(* PLC project test_IXL.project, CODESYS CODESYS V3.5 SP20 *)
(* stored: creationDateTime 2024-11-21T22:24:16.9503373, modificationDateTime 2024-07-08T19:29:50.2349361 *)

PROGRAM PLC_PRG
  VAR
    TC_occupied_101 : BOOL;
    TC_occupied_103 : BOOL;
    TC_occupied_105 : BOOL;
    TC_occupied_107 : BOOL;
    TC_occupied_109 : BOOL;
    TC_occupied_111 : BOOL;
    TC_occupied_113 : BOOL;
    TC_occupied_115 : BOOL;
    TC_occupied_102 : BOOL;
    TC_occupied_104 : BOOL;
    TC_occupied_106 : BOOL;
    TC_occupied_108 : BOOL;
    TC_occupied_110 : BOOL;
    TC_occupied_112 : BOOL;
    TC_occupied_114 : BOOL;
    TC_occupied_116 : BOOL;
    switch_detected_left_01 : BOOL;
    switch_detected_right_01 : BOOL;
    switch_detected_left_02 : BOOL;
    switch_detected_right_02 : BOOL;
    route_destruction_demand_AB : BOOL;
    route_destruction_demand_BC : BOOL;
    route_destruction_demand_ED : BOOL;
    route_destruction_demand_CD : BOOL;
    route_destruction_demand_DC : BOOL;
    route_destruction_demand_CB : BOOL;
    route_formation_demand_AB : BOOL;
    route_formation_demand_BC : BOOL;
    route_formation_demand_ED : BOOL;
    route_formation_demand_CD : BOOL;
    route_formation_demand_DC : BOOL;
    route_formation_demand_CB : BOOL;
    switch_manual_override_01 : BOOL;
    switch_manual_override_02 : BOOL;
    signal_open_route_201 : BOOL;
    signal_open_route_203 : BOOL;
    signal_open_route_205 : BOOL;
    signal_open_route_206 : BOOL;
    signal_open_route_208 : BOOL;
    signal_open_block_201 : BOOL;
    signal_open_block_203 : BOOL;
    signal_open_block_205 : BOOL;
    signal_open_block_206 : BOOL;
    signal_open_block_208 : BOOL;
    signal_open_block_207 : BOOL;
    signal_open_block_204 : BOOL;
    signal_open_block_210 : BOOL;
    switch_command_left_01 : BOOL;
    switch_command_right_01 : BOOL;
    switch_command_left_02 : BOOL;
    switch_command_right_02 : BOOL;
    route_open_AB : BOOL;
    route_open_BC : BOOL;
    route_open_ED : BOOL;
    route_open_CD : BOOL;
    route_open_DC : BOOL;
    route_open_CB : BOOL;
    route_destruction_acq_AB : BOOL;
    route_destruction_acq_BC : BOOL;
    route_destruction_acq_ED : BOOL;
    route_destruction_acq_CD : BOOL;
    route_destruction_acq_DC : BOOL;
    route_destruction_acq_CB : BOOL;
    route_state_AB : route_state;
    route_state_BC : route_state;
    route_state_ED : route_state;
    route_state_CD : route_state;
    route_state_DC : route_state;
    route_state_CB : route_state;
  END_VAR
  VAR CONSTANT
    DELAY_DEST_DC : TIME := TIME#30s0ms;
    DELAY_DEST_CB : TIME := TIME#30s0ms;
    DELAY_DEST_ED : TIME := TIME#30s0ms;
    DELAY_DEST_CD : TIME := TIME#30s0ms;
    DELAY_DEST_BC : TIME := TIME#30s0ms;
    DELAY_DEST_AB : TIME := TIME#30s0ms;
  END_VAR
  VAR
    direction_lock_CB : BOOL;
    direction_lock_AB : BOOL;
  END_VAR
  VAR  (* added by the conversion: wires and edge detectors of the diagram *)
    _AND70000000008_OUT : BOOL;
    _AND80000000007_OUT : BOOL;
  END_VAR

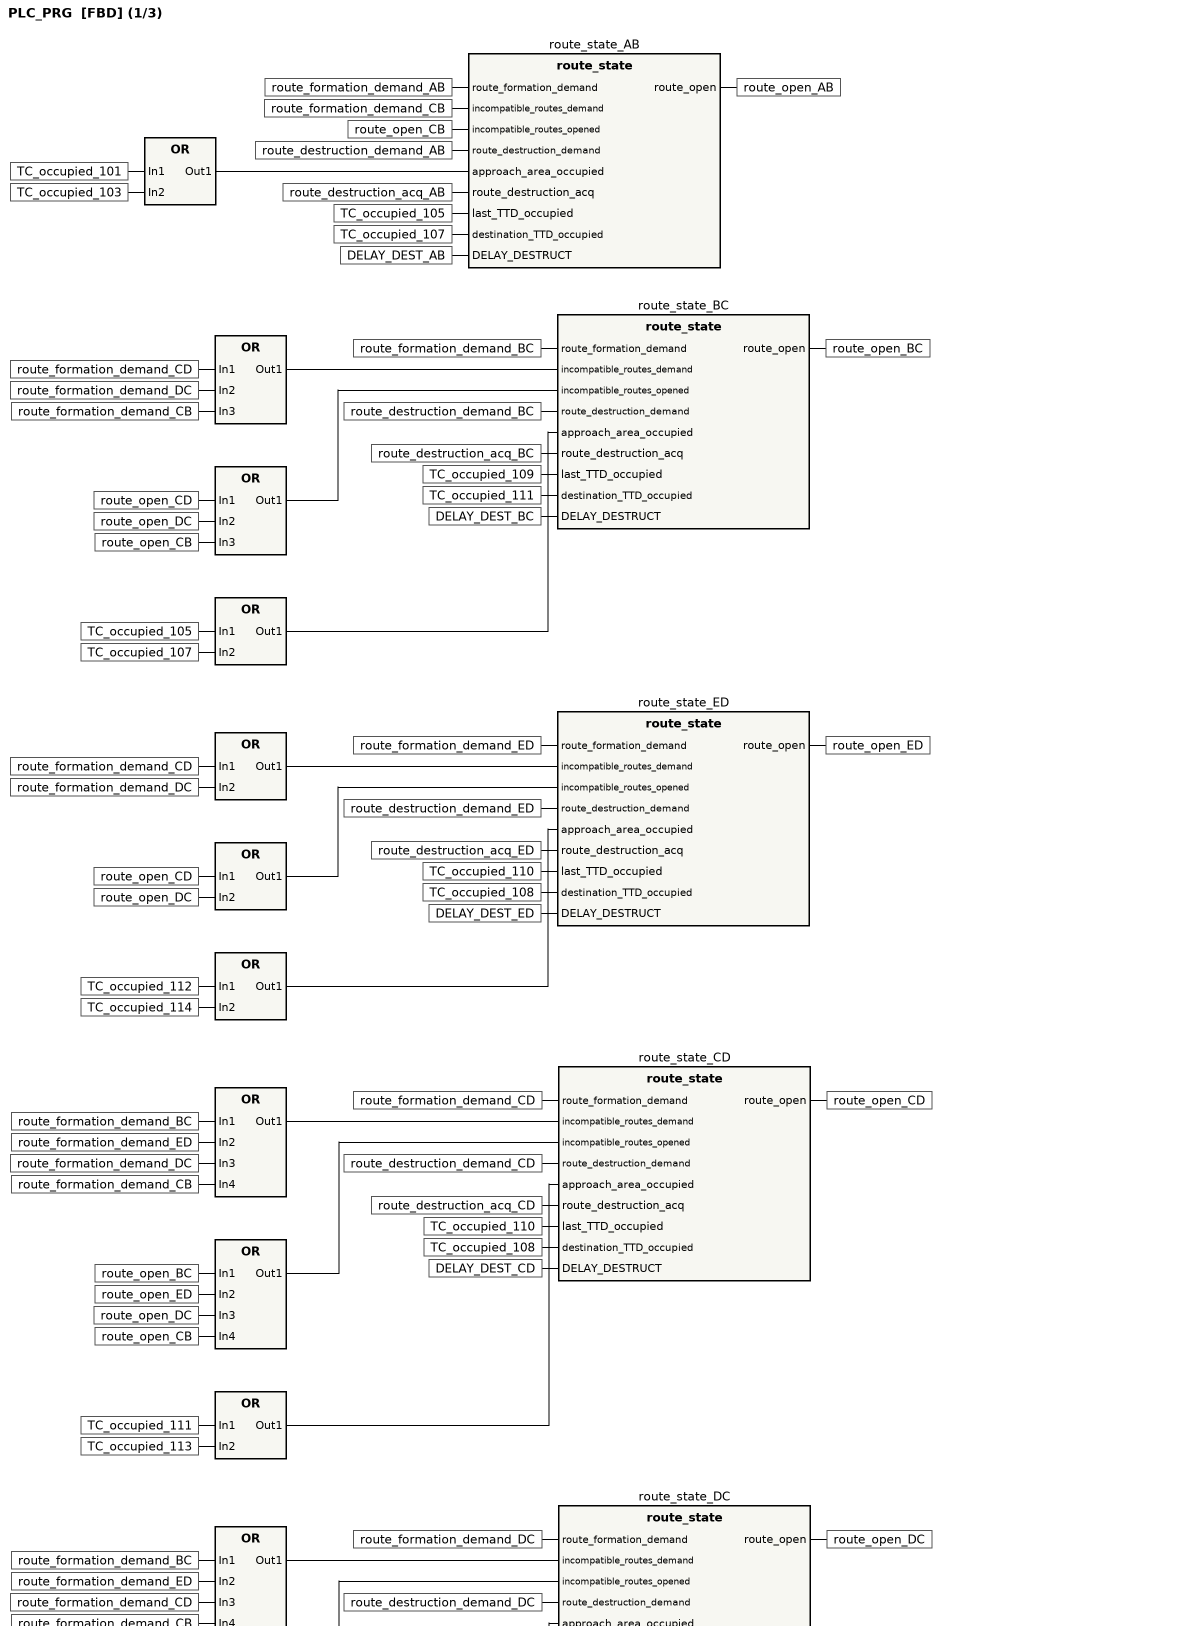
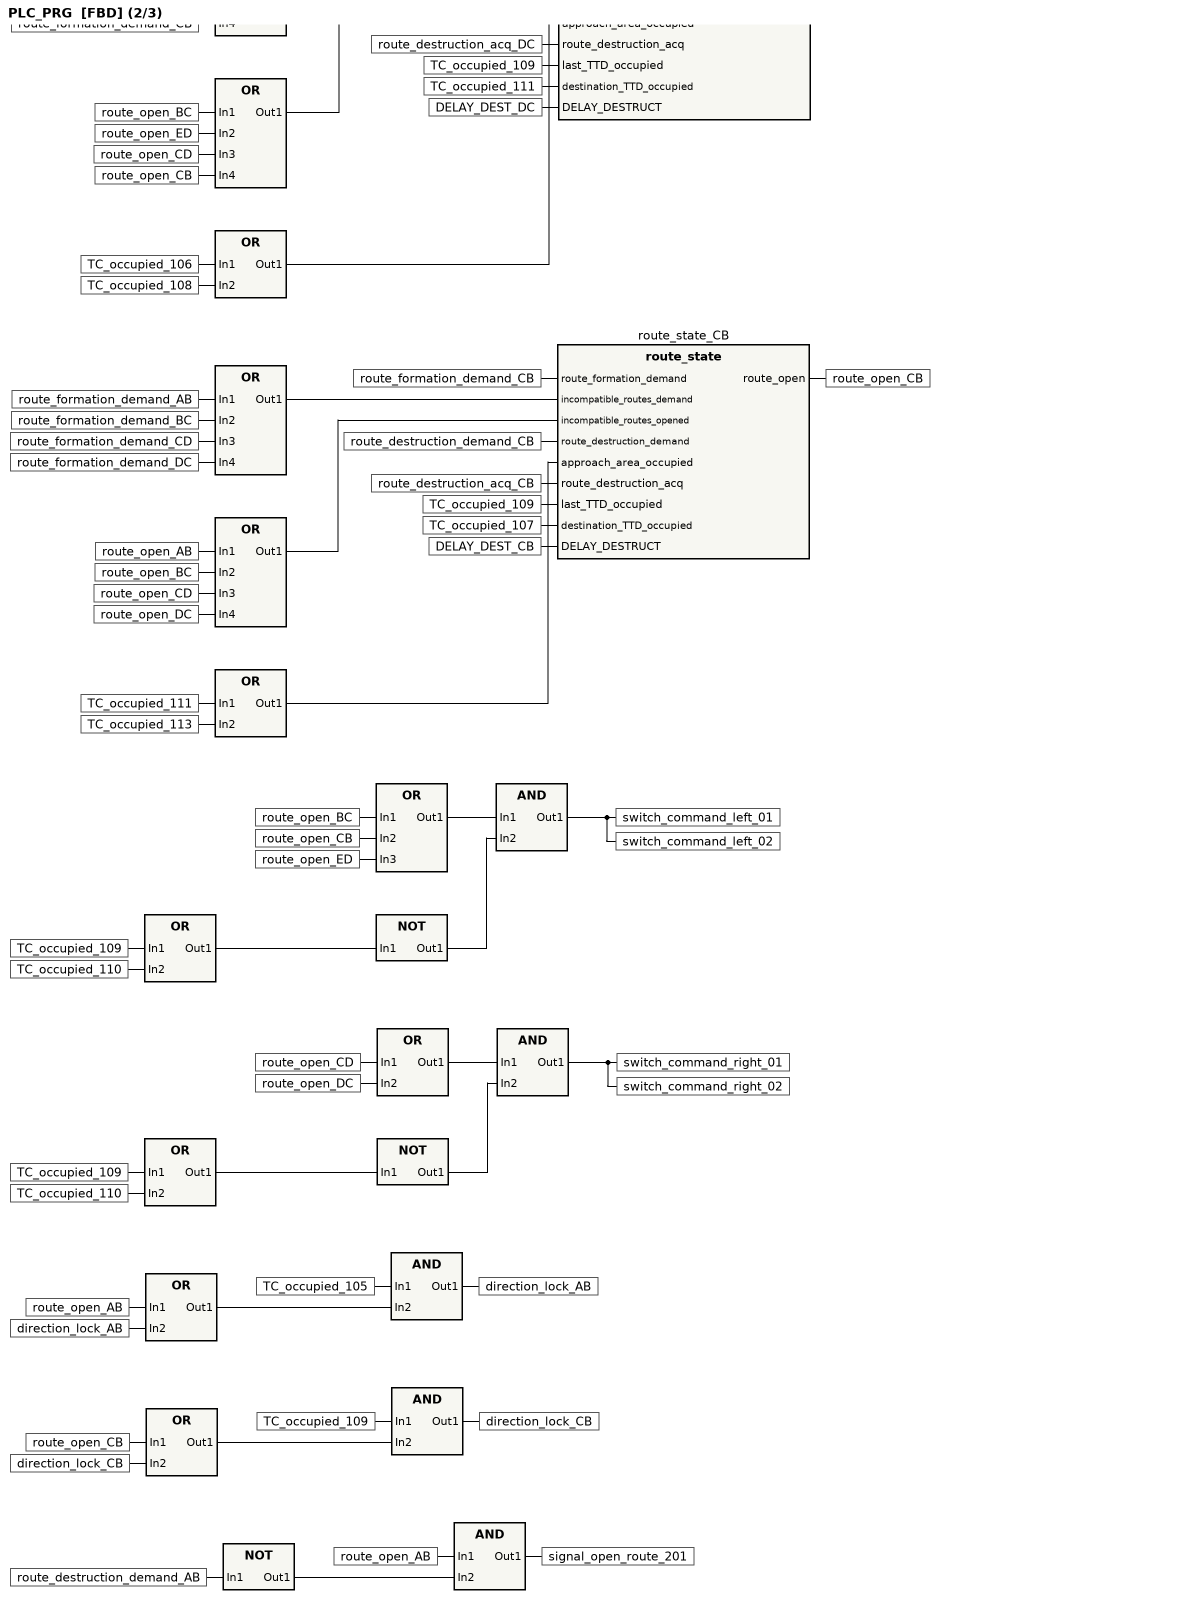
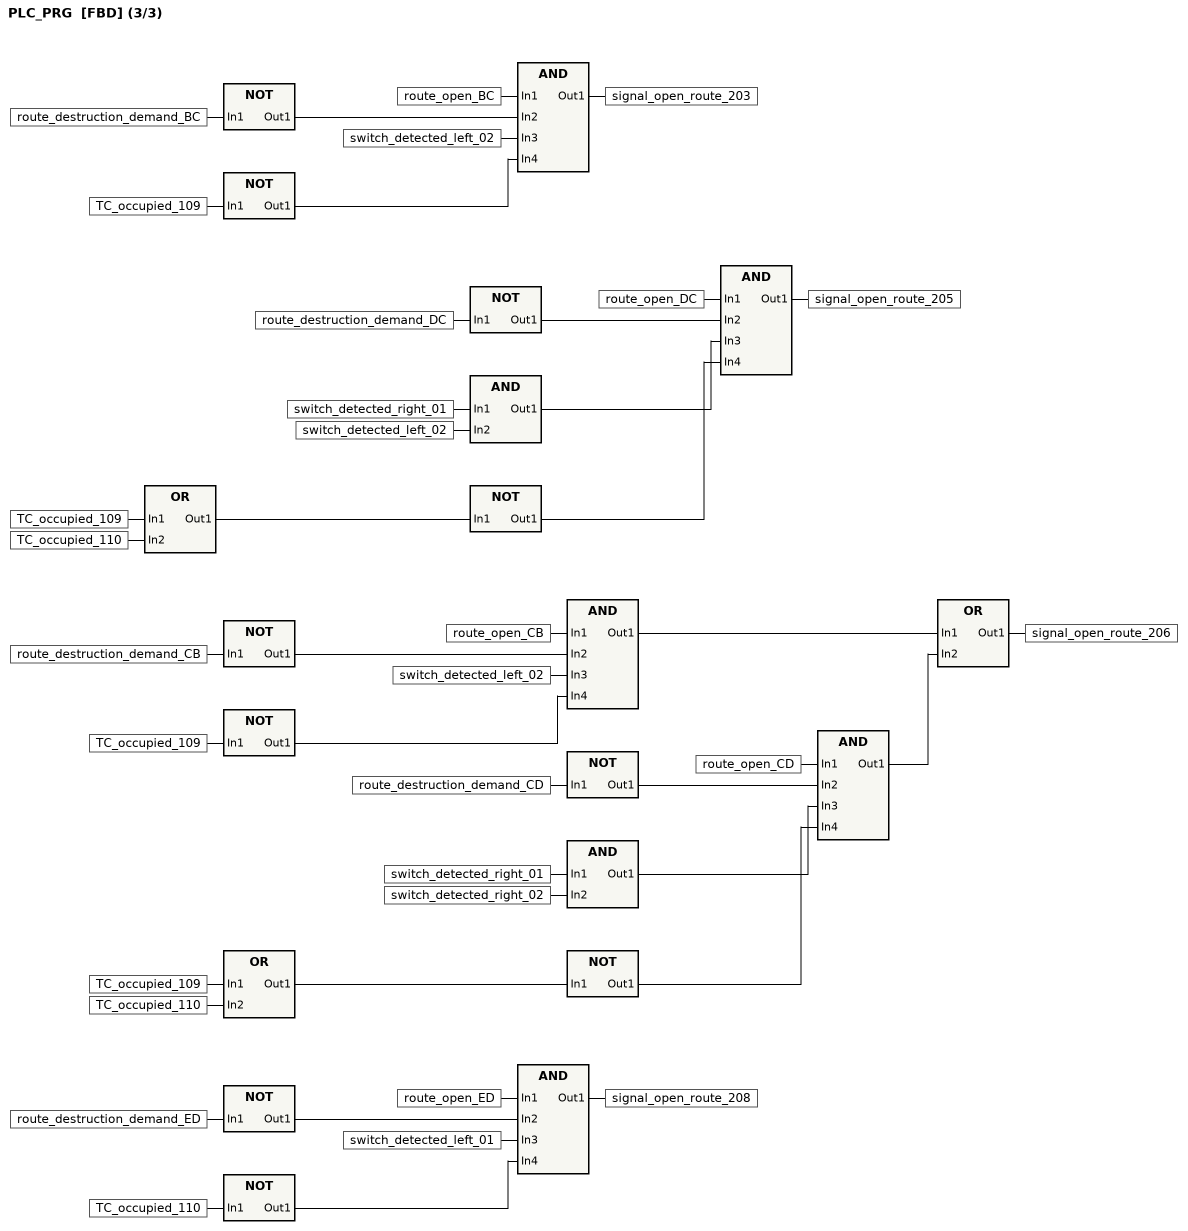
(* FBD diagram, written out as Structured Text *)
route_state_AB(route_formation_demand := route_formation_demand_AB, incompatible_routes_demand := route_formation_demand_CB, incompatible_routes_opened := route_open_CB, route_destruction_demand := route_destruction_demand_AB, approach_area_occupied := TC_occupied_101 OR TC_occupied_103, route_destruction_acq := route_destruction_acq_AB, last_TTD_occupied := TC_occupied_105, destination_TTD_occupied := TC_occupied_107, DELAY_DESTRUCT := DELAY_DEST_AB);
route_open_AB := route_state_AB.route_open;
route_state_BC(route_formation_demand := route_formation_demand_BC, incompatible_routes_demand := route_formation_demand_CD OR route_formation_demand_DC OR route_formation_demand_CB, incompatible_routes_opened := route_open_CD OR route_open_DC OR route_open_CB, route_destruction_demand := route_destruction_demand_BC, approach_area_occupied := TC_occupied_105 OR TC_occupied_107, route_destruction_acq := route_destruction_acq_BC, last_TTD_occupied := TC_occupied_109, destination_TTD_occupied := TC_occupied_111, DELAY_DESTRUCT := DELAY_DEST_BC);
route_open_BC := route_state_BC.route_open;
route_state_ED(route_formation_demand := route_formation_demand_ED, incompatible_routes_demand := route_formation_demand_CD OR route_formation_demand_DC, incompatible_routes_opened := route_open_CD OR route_open_DC, route_destruction_demand := route_destruction_demand_ED, approach_area_occupied := TC_occupied_112 OR TC_occupied_114, route_destruction_acq := route_destruction_acq_ED, last_TTD_occupied := TC_occupied_110, destination_TTD_occupied := TC_occupied_108, DELAY_DESTRUCT := DELAY_DEST_ED);
route_open_ED := route_state_ED.route_open;
route_state_CD(route_formation_demand := route_formation_demand_CD, incompatible_routes_demand := route_formation_demand_BC OR route_formation_demand_ED OR route_formation_demand_DC OR route_formation_demand_CB, incompatible_routes_opened := route_open_BC OR route_open_ED OR route_open_DC OR route_open_CB, route_destruction_demand := route_destruction_demand_CD, approach_area_occupied := TC_occupied_111 OR TC_occupied_113, route_destruction_acq := route_destruction_acq_CD, last_TTD_occupied := TC_occupied_110, destination_TTD_occupied := TC_occupied_108, DELAY_DESTRUCT := DELAY_DEST_CD);
route_open_CD := route_state_CD.route_open;
route_state_DC(route_formation_demand := route_formation_demand_DC, incompatible_routes_demand := route_formation_demand_BC OR route_formation_demand_ED OR route_formation_demand_CD OR route_formation_demand_CB, incompatible_routes_opened := route_open_BC OR route_open_ED OR route_open_CD OR route_open_CB, route_destruction_demand := route_destruction_demand_DC, approach_area_occupied := TC_occupied_106 OR TC_occupied_108, route_destruction_acq := route_destruction_acq_DC, last_TTD_occupied := TC_occupied_109, destination_TTD_occupied := TC_occupied_111, DELAY_DESTRUCT := DELAY_DEST_DC);
route_open_DC := route_state_DC.route_open;
route_state_CB(route_formation_demand := route_formation_demand_CB, incompatible_routes_demand := route_formation_demand_AB OR route_formation_demand_BC OR route_formation_demand_CD OR route_formation_demand_DC, incompatible_routes_opened := route_open_AB OR route_open_BC OR route_open_CD OR route_open_DC, route_destruction_demand := route_destruction_demand_CB, approach_area_occupied := TC_occupied_111 OR TC_occupied_113, route_destruction_acq := route_destruction_acq_CB, last_TTD_occupied := TC_occupied_109, destination_TTD_occupied := TC_occupied_107, DELAY_DESTRUCT := DELAY_DEST_CB);
route_open_CB := route_state_CB.route_open;
_AND70000000008_OUT := (route_open_BC OR route_open_CB OR route_open_ED) AND NOT (TC_occupied_109 OR TC_occupied_110);
switch_command_left_01 := _AND70000000008_OUT;
switch_command_left_02 := _AND70000000008_OUT;
_AND80000000007_OUT := (route_open_CD OR route_open_DC) AND NOT (TC_occupied_109 OR TC_occupied_110);
switch_command_right_01 := _AND80000000007_OUT;
switch_command_right_02 := _AND80000000007_OUT;
direction_lock_AB := TC_occupied_105 AND (route_open_AB OR direction_lock_AB);
direction_lock_CB := TC_occupied_109 AND (route_open_CB OR direction_lock_CB);
signal_open_route_201 := route_open_AB AND NOT route_destruction_demand_AB;
signal_open_route_203 := route_open_BC AND NOT route_destruction_demand_BC AND switch_detected_left_02 AND NOT TC_occupied_109;
signal_open_route_205 := route_open_DC AND NOT route_destruction_demand_DC AND switch_detected_right_01 AND switch_detected_left_02 AND NOT (TC_occupied_109 OR TC_occupied_110);
signal_open_route_206 := route_open_CB AND NOT route_destruction_demand_CB AND switch_detected_left_02 AND NOT TC_occupied_109 OR route_open_CD AND NOT route_destruction_demand_CD AND switch_detected_right_01 AND switch_detected_right_02 AND NOT (TC_occupied_109 OR TC_occupied_110);
signal_open_route_208 := route_open_ED AND NOT route_destruction_demand_ED AND switch_detected_left_01 AND NOT TC_occupied_110;
END_PROGRAM

{attribute 'do_checks_for_implicit_code'}
FUNCTION_BLOCK AUTO_DESTRUCT
  VAR_INPUT
    route_state : BOOL;
    last_TTD_occupied : BOOL;
    destination_TTD_occupied : BOOL;
  END_VAR
  VAR_OUTPUT
    route_auto_destruc_command : BOOL;
  END_VAR

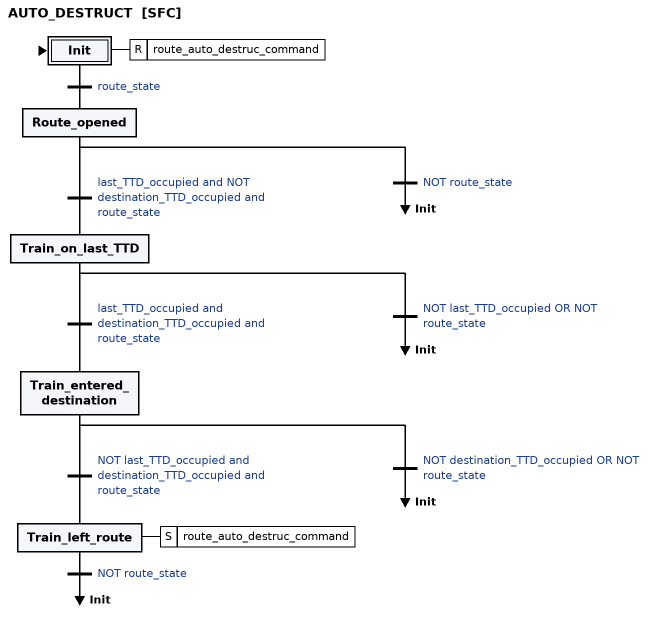
INITIAL_STEP Init:
  route_auto_destruc_command(R);
END_STEP
TRANSITION FROM Init TO Route_opened
  := route_state;
END_TRANSITION
STEP Route_opened:
END_STEP
TRANSITION FROM Route_opened TO Train_on_last_TTD
  := last_TTD_occupied and NOT destination_TTD_occupied and route_state;
END_TRANSITION
TRANSITION FROM Route_opened TO Init
  := NOT route_state;
END_TRANSITION
STEP Train_on_last_TTD:
END_STEP
TRANSITION FROM Train_on_last_TTD TO Train_entered_destination
  := last_TTD_occupied and destination_TTD_occupied and route_state;
END_TRANSITION
TRANSITION FROM Train_on_last_TTD TO Init
  := NOT last_TTD_occupied OR NOT route_state;
END_TRANSITION
STEP Train_entered_destination:
END_STEP
TRANSITION FROM Train_entered_destination TO Train_left_route
  := NOT last_TTD_occupied and destination_TTD_occupied and route_state;
END_TRANSITION
TRANSITION FROM Train_entered_destination TO Init
  := NOT destination_TTD_occupied OR NOT route_state;
END_TRANSITION
STEP Train_left_route:
  route_auto_destruc_command(S);
END_STEP
TRANSITION FROM Train_left_route TO Init
  := NOT route_state;
END_TRANSITION
END_FUNCTION_BLOCK

FUNCTION_BLOCK route_state
  VAR_INPUT
    route_formation_demand : BOOL;
    incompatible_routes_demand : BOOL;
    incompatible_routes_opened : BOOL;
    route_destruction_demand : BOOL;
    approach_area_occupied : BOOL;
    route_destruction_acq : BOOL;
    last_TTD_occupied : BOOL;
    destination_TTD_occupied : BOOL;
    {attribute 'input_constant'}
    DELAY_DESTRUCT : TIME;
  END_VAR
  VAR_OUTPUT
    route_open : BOOL;
  END_VAR
  VAR
    SR_route : SR;
    Auto_destruct_state_machine : AUTO_DESTRUCT;
    TON_manual_destruct : TON;
  END_VAR

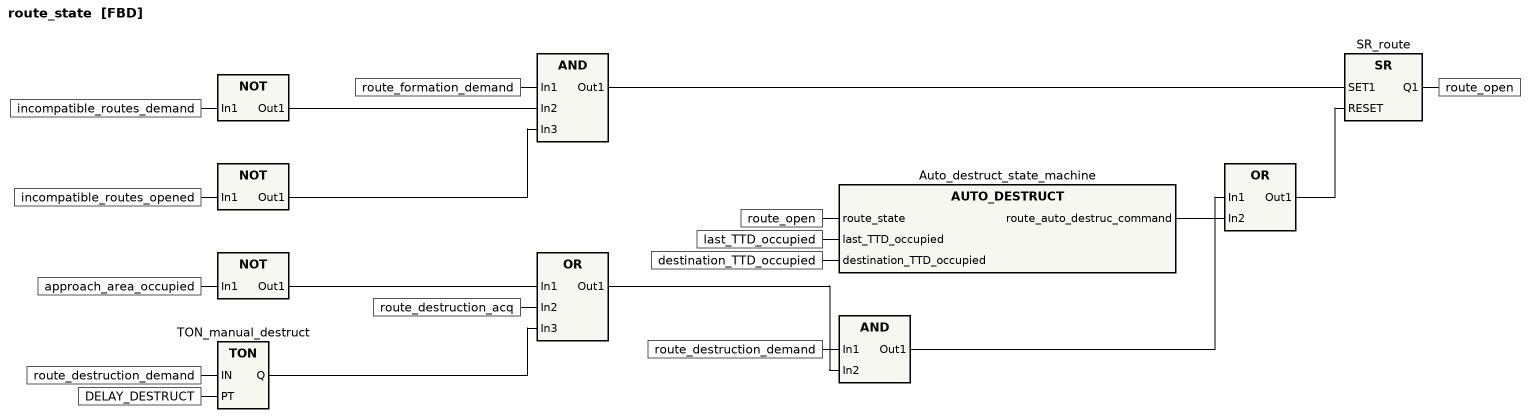
(* FBD diagram, written out as Structured Text *)
TON_manual_destruct(IN := route_destruction_demand, PT := DELAY_DESTRUCT);
Auto_destruct_state_machine(route_state := route_open, last_TTD_occupied := last_TTD_occupied, destination_TTD_occupied := destination_TTD_occupied);
SR_route(SET1 := route_formation_demand AND NOT incompatible_routes_demand AND NOT incompatible_routes_opened, RESET := route_destruction_demand AND (NOT approach_area_occupied OR route_destruction_acq OR TON_manual_destruct.Q) OR Auto_destruct_state_machine.route_auto_destruc_command);
route_open := SR_route.Q1;
END_FUNCTION_BLOCK

CONFIGURATION Device
  RESOURCE Application ON PLC
    TASK MainTask(INTERVAL := T#20ms, PRIORITY := 1);
    PROGRAM PLC_PRG WITH MainTask : PLC_PRG;
  END_RESOURCE
END_CONFIGURATION
